// TIA Portal V21 export
TYPE "AxixAS_DataIn_Type_v2.0"
   STRUCT
      ixEnablePos { S7_SetPoint := 'True'} : Bool;   // Enable positioner / Abilita asse
      ixDriveReady { S7_SetPoint := 'True'} : Bool;   // Inverter magnetizzato
      ixEnableLevRes { S7_SetPoint := 'True'} : Bool;   // Enable level research / Abilita ricerca livello
      ixLevelReached { S7_SetPoint := 'True'} : Bool;   // = 1 Sensore livello raggiunto
      ixMotorReadyReq { S7_SetPoint := 'True'} : Bool;   // Richiede magnetizzazione Motore
      ixAlarmReset { S7_SetPoint := 'True'} : Bool;   // Reset alarms / Reset allarmi
      ixAbort { S7_SetPoint := 'True'} : Bool;   // Initializing motor encoder position / Abort sistema
      ixJogPos { S7_SetPoint := 'True'} : Bool;   // Manual Jog positive / Manuale JOG +
      ixJogNeg { S7_SetPoint := 'True'} : Bool;   // Manual Jog negative / Manuale JOG -
      xAutoSpeedDetect { S7_SetPoint := 'True'} : Bool;   // Calcolo velocità automatico su movimento
      xAutoAccDecCalculation { S7_SetPoint := 'True'} : Bool;   // Calcolo Acc Dec automatico su velocità
      ifPositionRequest { S7_SetPoint := 'True'} : Real;   // Position requested (mm) / Quota richiesta (mm)
      ifSpeedRequest { S7_SetPoint := 'True'} : Real;   // Speed requested (mm/sec) / Velocità richiesta (mm/sec)
      ifPositionStartLev { S7_SetPoint := 'True'} : Real;   // Position start research (mm) / Quota inizio ricerca (mm)
      ifSpeedLev { S7_SetPoint := 'True'} : Real;   // Research speed (mm/sec) / Velocità ricerca (mm/sec)
      ifAccRamp { S7_SetPoint := 'True'} : Real;   // Acceleration ramp (mm/sec^2) / * Rampa accelerazione (mm/sec^2)
      ifDecRamp { S7_SetPoint := 'True'} : Real;   // Deceleration ramp (mm/sec^2) / * Rampa decelerazione (mm/sec^2)
      ifTimeScan { S7_SetPoint := 'True'} : Real;   // Time last scan (sec) / Tempo ultima scansione (sec)
      ifEncoder { S7_SetPoint := 'True'} : Real;   // Actual encoder position (encoder) / Posizione attuale encoder
   END_STRUCT;
END_TYPE
